FUNCTION WithinRange : BOOL
VAR_INPUT
    ValA	:	REAL; //New position to evaluate
    Center :	REAL; //Current position
    Range : REAL; //Span of the range
    Offset	:	REAL := 0; //Offset from center if the range is non-symetric
END_VAR
VAR
END_VAR

IF ValA < (Center + Offset - (Range/2) ) THEN
    WithinRange := FALSE;
ELSIF ValA > (Center + Offset + (Range/2) ) THEN
    WithinRange := FALSE;
ELSE
    WithinRange := TRUE;
END_IF

END_FUNCTION

(* stored: Version 1.1.0.1, ProductVersion 3.1.4022.18
   POU WithinRange: Id {665d2067-503e-41d4-add4-3ba7efc451a5}, SpecialFunc None *)
